TYPE Position :
STRUCT
	Axis : INT;
	Distance : LREAL;
	
END_STRUCT
END_TYPE

(* stored: Version 1.1.0.1, ProductVersion 3.1.4024.14
   DUT Position: Id {9e75f1b8-2bc4-4206-b555-92bb44116cf9} *)
